Universal Robots PolyScope program: translation_sample_servoj.urp

Program translation_sample_servoj (installation=EE no fingers directory=/programs/daniel_rtde createdIn=3.2.19275.0 lastSavedIn=5.8.0.10253 robotSerialNumber=20205501313)
Calibrated DH parameters: a=[-0.000005, -0.295085, -0.38277, -0.000042, 0.000047, 0]; d=[0.162617, -370.906238, 381.183803, -10.144133, 0.099913, 0.099543]; alpha=[1.571245, -0.000826, 0.008484, 1.571183, -1.570198, 0]; deltaTheta=[0, 0.803921, 5.703226, -0.223968, 0, 0]
BeforeStart
  joints := get_actual_joint_positions()
  Script: write_output_boolean_register(0, False )
  Wait Sleep waitTime=0.01
  Script: popup("Registers reset, run PC code and then click Continue",title="Hi Daniel",blocking= True )
  mode := 0
Robot Program (runOnlyOnce=false)
  Script: write_output_boolean_register(0, True )
  Script: sync()
  Loop While (checkContinuously=false) expression=mode<3
    Loop While (checkContinuously=false) expression=mode≟1
      MoveJ speed 60 deg/s, acceleration 80 deg/s^2 (useActiveTCP=true) feature=Base
        Waypoint Waypoint (Variable): variable(name=joints)
      Script: write_output_boolean_register(0, False )
      Script: sync()
    Loop While (checkContinuously=false) expression=mode≟2
      Script: servoj(joints, 0, 0, 0.002, 0.2, 2000)
    Loop While (checkContinuously=false) expression=mode≟3
      Halt
  Script: sync()
Thread Thread_1 (runOnlyOnce=false)
  tmp := p[0,0,0,0,0,0]
  Loop Forever
    Script file /programs/pose_register.script
      | tmp[0]=read_input_float_register(0)
      | tmp[1]=read_input_float_register(1)
      | tmp[2]=read_input_float_register(2)
      | tmp[3]=read_input_float_register(3)
      | tmp[4]=read_input_float_register(4)
      | tmp[5]=read_input_float_register(5)
    joints := get_inverse_kin(p[tmp[0],tmp[1],tmp[2],tmp[3],tmp[4],tmp[5]],get_actual_joint_positions())
    Script: sync()
    mode := read_input_integer_register(0)
    Script: sync()
